// Block: PPrgArchive13

DATA_BLOCK PPrgArchive13
VERSION : 0.1
   NON_RETAIN
   VAR
      PRG : Array[1201..1300] of PPrg_Data;
   END_VAR

BEGIN
   // No initialization required
END_DATA_BLOCK
